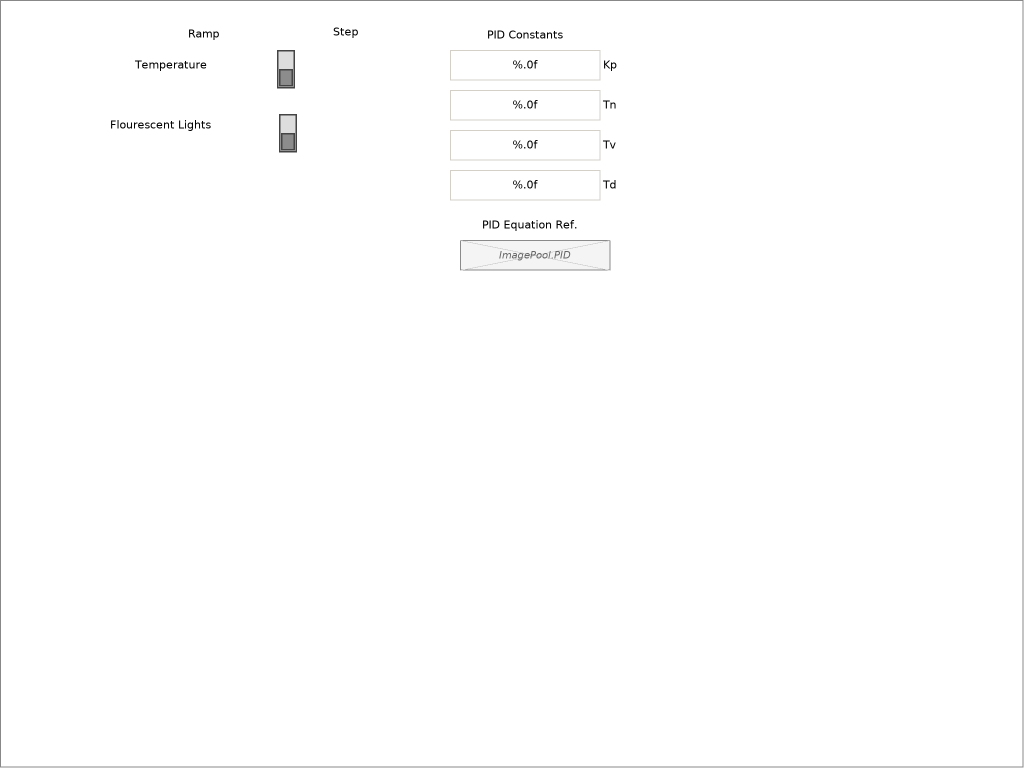
VISUALIZATION Settings  // 1024x768
    DipSwitch (251,50 70x38), variable: GVL.TempStepmode, behaviour: TOGGLE, style: Switch-DipSwitch-Gray
    DipSwitch (253,114 70x38), variable: GVL.Light1Stepmode, behaviour: TOGGLE, style: Switch-DipSwitch-Gray
    Label (10,50 200x30), "Temperature"
    Label (14,110 200x30), "Flourescent Lights"
    Label (185,19 67x30), "Ramp"
    Label (330,18 49x28), "Step"
    Textfield (450,50 150x30), "%.0f", text variable: GVL.KpCooling
        OnMouseClick: write the text variable via VisuDialogs.Numpad, min 0
    Textfield (450,90 150x30), "%.0f", text variable: GVL.KiCooling
        OnMouseClick: write the text variable via VisuDialogs.Numpad, min 0
    Textfield (450,130 150x30), "%.0f", text variable: GVL.KvCooling
        OnMouseClick: write the text variable via VisuDialogs.Numpad, min 0
    Label (600,50 30x30), "Kp"
    Label (600,90 30x30), "Tn"
    Label (600,130 30x30), "Tv"
    Image (460,240 150x30), image: ImagePool.PID
    Textfield (450,170 150x30), "%.0f", text variable: GVL.KdCooling
        OnMouseClick: write the text variable via VisuDialogs.Numpad, min 0
    Label (600,170 30x30), "Td"
    Label (450,20 150x30), "PID Constants"
    Label (430,210 200x30), "PID Equation Ref."
END_VISUALIZATION

(* stored: Version 1.1.0.1, ProductVersion 3.1.4022.18
   Visu Settings: Id {1b33a30b-6a18-49e6-aec2-86545f52a8b5} *)
